# EPICS autosave request: motorApp/Db/trajectoryScan_settings.req
$(P)$(R)Nelements
$(P)$(R)MoveMode
$(P)$(R)Npulses
$(P)$(R)StartPulses
$(P)$(R)EndPulses
$(P)$(R)TimeMode
$(P)$(R)Time
$(P)$(R)TimeScale
$(P)$(R)Accel
$(P)$(R)TrajectoryFile
$(P)$(R)DebugLevel
$(P)$(R)M1Move
$(P)$(R)M2Move
$(P)$(R)M3Move
$(P)$(R)M4Move
$(P)$(R)M5Move
$(P)$(R)M6Move
$(P)$(R)M7Move
$(P)$(R)M8Move
$(P)$(R)SimMode
$(P)$(R)TimeTraj
$(P)$(R)M1Traj
$(P)$(R)M2Traj
$(P)$(R)M3Traj
$(P)$(R)M4Traj
$(P)$(R)M5Traj
$(P)$(R)M6Traj
$(P)$(R)M7Traj
$(P)$(R)M8Traj

# MAX controller specific
$(P)$(R)realTimeTrajectory
$(P)$(R)OutBitNum
$(P)$(R)InBitNum
$(P)$(R)OverrideFactor
$(P)$(R)UpdateFreq
$(P)$(R)M1MinSpeed
$(P)$(R)M2MinSpeed
$(P)$(R)M3MinSpeed
$(P)$(R)M4MinSpeed
$(P)$(R)M5MinSpeed
$(P)$(R)M6MinSpeed
$(P)$(R)M7MinSpeed
$(P)$(R)M8MinSpeed
$(P)$(R)M1MaxSpeed
$(P)$(R)M2MaxSpeed
$(P)$(R)M3MaxSpeed
$(P)$(R)M4MaxSpeed
$(P)$(R)M5MaxSpeed
$(P)$(R)M6MaxSpeed
$(P)$(R)M7MaxSpeed
$(P)$(R)M8MaxSpeed
$(P)$(R)AddAccelDecel
$(P)$(R)PulseDir
$(P)$(R)PulseLenUS
$(P)$(R)PulseSrc
$(P)$(R)PulseMode
$(P)$(R)PulsePositions
